PROGRAM Anlage
VAR_INPUT
	UR5				:FB_Roboter;
	Gripper			:FB_SmartGreifer;
	HEX_E_V2		:FB_Kraftsensor_V2;
END_VAR

VAR
END_VAR

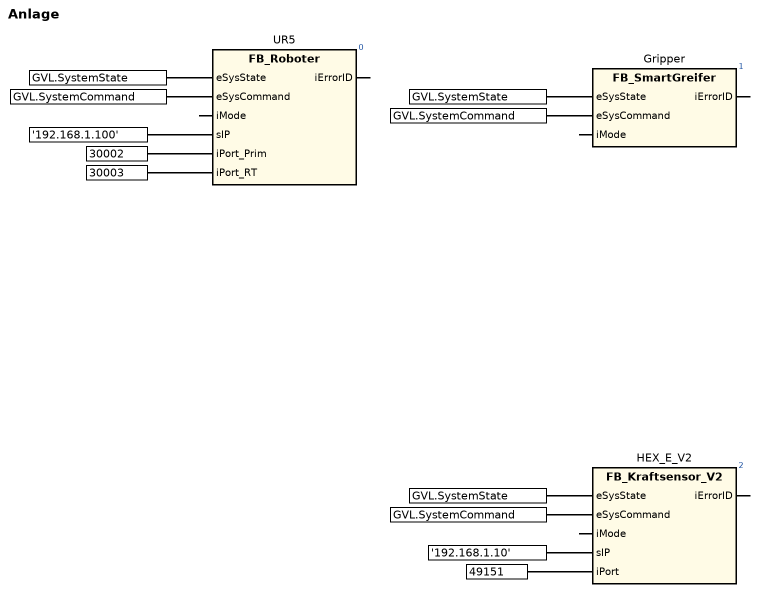
UR5(
    eSysState := GVL.SystemState,
    eSysCommand := GVL.SystemCommand,
    sIP := '192.168.1.100',
    iPort_Prim := 30002,
    iPort_RT := 30003); // FB_Roboter
Gripper(eSysState := GVL.SystemState, eSysCommand := GVL.SystemCommand); // FB_SmartGreifer
HEX_E_V2(
    eSysState := GVL.SystemState,
    eSysCommand := GVL.SystemCommand,
    sIP := '192.168.1.10',
    iPort := 49151); // FB_Kraftsensor_V2

END_PROGRAM

(* stored: Version 1.1.0.1
   POU Anlage: Id {c0949e1e-582a-4e6c-80fc-b378d417eaa8}, SpecialFunc None *)
